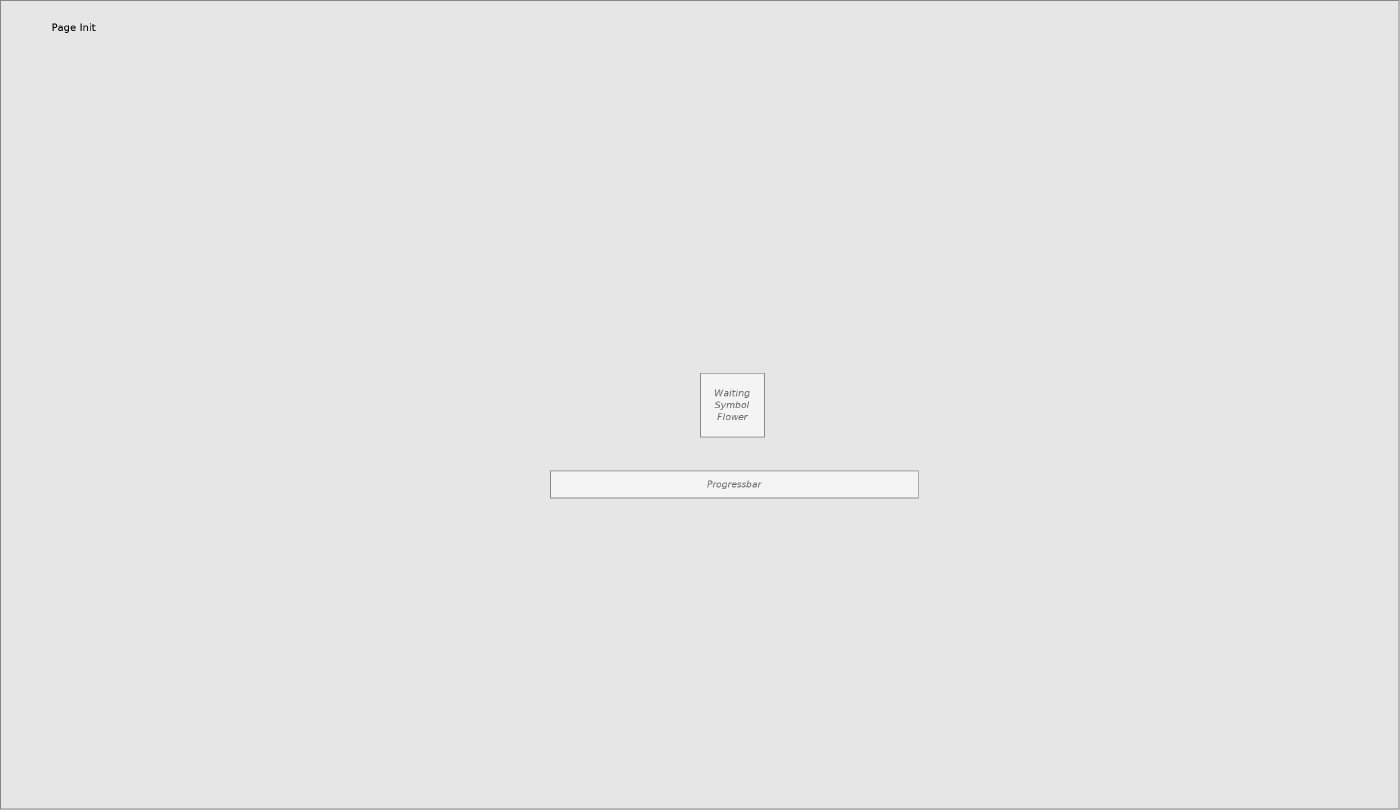
VISUALIZATION PageInitializing  // 1520x880
VAR_IN_OUT
	iProgressBar : USINT;
END_VAR
    Progressbar (597,511 400x30), variable: iProgressBar
    WaitingSymbolFlower (760,405 70x70)
    Label (5,15 150x30), "Page Init"
END_VISUALIZATION

(* stored: Version 1.1.0.1, ProductVersion 3.1.4024.9
   Visu PageInitializing: Id {abc60465-2b7b-4887-a728-03f417e9af64} *)
